// TIA Portal V16 export
// export: Created 2021-11-12T13:33:14.2128185Z, ExportSetting WithDefaults, DisplayName Totally Integrated Automation Portal, DisplayVersion V16 Update 3, DisplayName TIA Portal Version Control Interface, DisplayVersion V16 Update 2, DisplayName TIA Portal Openness, DisplayVersion V16 Update 3, DisplayName SINAMICS Startdrive Advanced, DisplayVersion V16 Update 5, DisplayName SINAMICS Startdrive G130, G150, S120, S150, SINAMICS MV, S210, DisplayVersion V16 Update 5, DisplayName SINAMICS Startdrive G110M, G120, G120C, G120D, G120P, G115D, DisplayVersion V16 Update 5, DisplayName STEP 7 Professional, DisplayVersion V16 Update 3, DisplayName STEP 7 Safety, DisplayVersion V16, DisplayName WinCC UA Professional, DisplayVersion V16 Update 3
FUNCTION_BLOCK "IM_400+UH31-KF10"   // FB24, LAD
TITLE = Inputs reading
{ S7_Optimized_Access := 'TRUE' }
VERSION : 0.1
// MICE Wood interface block
// stored: AutoNumber true, IsIECCheckEnabled false, IsRetainMemResEnabled false, MemoryReserve 100, SetENOAutomatically false, UDAEnableTagReadback false
   VAR
      KF11_Ix0 { S7_SetPoint := 'True'} : "STD_CH_DI";
      KF11_Ix1 { S7_SetPoint := 'True'} : "STD_CH_DI";
      KF11_Ix2 { S7_SetPoint := 'True'} : "STD_CH_DI";
      KF11_Ix3 { S7_SetPoint := 'True'} : "STD_CH_DI";
      KF11_Ix4 { S7_SetPoint := 'True'} : "STD_CH_DI";
      KF11_Ix5 { S7_SetPoint := 'True'} : "STD_CH_DI";
      KF11_Ix6 { S7_SetPoint := 'True'} : "STD_CH_DI";
      KF11_Ix7 { S7_SetPoint := 'True'} : "STD_CH_DI";
      KF12_Ix0 { S7_SetPoint := 'True'} : "STD_CH_DI";
      KF12_Ix1 { S7_SetPoint := 'True'} : "STD_CH_DI";
      KF12_Ix2 { S7_SetPoint := 'True'} : "STD_CH_DI";
      KF12_Ix3 { S7_SetPoint := 'True'} : "STD_CH_DI";
      KF12_Ix4 { S7_SetPoint := 'True'} : "STD_CH_DI";
      KF12_Ix5 { S7_SetPoint := 'True'} : "STD_CH_DI";
      KF12_Ix6 { S7_SetPoint := 'True'} : "STD_CH_DI";
      KF12_Ix7 { S7_SetPoint := 'True'} : "STD_CH_DI";
      KF12_Ix8 { S7_SetPoint := 'True'} : "STD_CH_DI";
      KF12_Ix9 { S7_SetPoint := 'True'} : "STD_CH_DI";
      KF12_Ix10 { S7_SetPoint := 'True'} : "STD_CH_DI";
      KF12_Ix11 { S7_SetPoint := 'True'} : "STD_CH_DI";
      KF12_Ix12 { S7_SetPoint := 'True'} : "STD_CH_DI";
      KF12_Ix13 { S7_SetPoint := 'True'} : "STD_CH_DI";
      KF12_Ix14 { S7_SetPoint := 'True'} : "STD_CH_DI";
      KF12_Ix15 { S7_SetPoint := 'True'} : "STD_CH_DI";
      KF13_Ix0 { S7_SetPoint := 'True'} : "STD_CH_DI";
      KF13_Ix1 { S7_SetPoint := 'True'} : "STD_CH_DI";
      KF13_Ix2 { S7_SetPoint := 'True'} : "STD_CH_DI";
      KF13_Ix3 { S7_SetPoint := 'True'} : "STD_CH_DI";
      KF13_Ix4 { S7_SetPoint := 'True'} : "STD_CH_DI";
      KF13_Ix5 { S7_SetPoint := 'True'} : "STD_CH_DI";
      KF13_Ix6 { S7_SetPoint := 'True'} : "STD_CH_DI";
      KF13_Ix7 { S7_SetPoint := 'True'} : "STD_CH_DI";
      KF13_Ix8 { S7_SetPoint := 'True'} : "STD_CH_DI";
      KF13_Ix9 { S7_SetPoint := 'True'} : "STD_CH_DI";
      KF13_Ix10 { S7_SetPoint := 'True'} : "STD_CH_DI";
      KF13_Ix11 { S7_SetPoint := 'True'} : "STD_CH_DI";
      KF13_Ix12 { S7_SetPoint := 'True'} : "STD_CH_DI";
      KF13_Ix13 { S7_SetPoint := 'True'} : "STD_CH_DI";
      KF13_Ix14 { S7_SetPoint := 'True'} : "STD_CH_DI";
      KF13_Ix15 { S7_SetPoint := 'True'} : "STD_CH_DI";
      KF14_Ix0 { S7_SetPoint := 'True'} : "STD_CH_DI";
      KF14_Ix1 { S7_SetPoint := 'True'} : "STD_CH_DI";
      KF14_Ix2 { S7_SetPoint := 'True'} : "STD_CH_DI";
      KF14_Ix3 { S7_SetPoint := 'True'} : "STD_CH_DI";
      KF14_Ix4 { S7_SetPoint := 'True'} : "STD_CH_DI";
      KF14_Ix5 { S7_SetPoint := 'True'} : "STD_CH_DI";
      KF14_Ix6 { S7_SetPoint := 'True'} : "STD_CH_DI";
      KF14_Ix7 { S7_SetPoint := 'True'} : "STD_CH_DI";
      KF14_Ix8 { S7_SetPoint := 'True'} : "STD_CH_DI";
      KF14_Ix9 { S7_SetPoint := 'True'} : "STD_CH_DI";
      KF14_Ix10 { S7_SetPoint := 'True'} : "STD_CH_DI";
      KF14_Ix11 { S7_SetPoint := 'True'} : "STD_CH_DI";
      KF14_Ix12 { S7_SetPoint := 'True'} : "STD_CH_DI";
      KF14_Ix13 { S7_SetPoint := 'True'} : "STD_CH_DI";
      KF14_Ix14 { S7_SetPoint := 'True'} : "STD_CH_DI";
      KF14_Ix15 { S7_SetPoint := 'True'} : "STD_CH_DI";
      KF15_Ix0 { S7_SetPoint := 'True'} : "STD_CH_DI";
      KF15_Ix1 { S7_SetPoint := 'True'} : "STD_CH_DI";
      KF15_Ix2 { S7_SetPoint := 'True'} : "STD_CH_DI";
      KF15_Ix3 { S7_SetPoint := 'True'} : "STD_CH_DI";
      KF15_Ix4 { S7_SetPoint := 'True'} : "STD_CH_DI";
      KF15_Ix5 { S7_SetPoint := 'True'} : "STD_CH_DI";
      KF15_Ix6 { S7_SetPoint := 'True'} : "STD_CH_DI";
      KF15_Ix7 { S7_SetPoint := 'True'} : "STD_CH_DI";
      KF15_Ix8 { S7_SetPoint := 'True'} : "STD_CH_DI";
      KF15_Ix9 { S7_SetPoint := 'True'} : "STD_CH_DI";
      KF15_Ix10 { S7_SetPoint := 'True'} : "STD_CH_DI";
      KF15_Ix11 { S7_SetPoint := 'True'} : "STD_CH_DI";
      KF15_Ix12 { S7_SetPoint := 'True'} : "STD_CH_DI";
      KF15_Ix13 { S7_SetPoint := 'True'} : "STD_CH_DI";
      KF15_Ix14 { S7_SetPoint := 'True'} : "STD_CH_DI";
      KF15_Ix15 { S7_SetPoint := 'True'} : "STD_CH_DI";
      KF61_AI0 { S7_SetPoint := 'True'} : "STD_CH_AI";
      KF61_AI1 { S7_SetPoint := 'True'} : "STD_CH_AI";
      KF61_AI2 { S7_SetPoint := 'True'} : "STD_CH_AI";
      KF61_AI3 { S7_SetPoint := 'True'} : "STD_CH_AI";
   END_VAR
   VAR_TEMP   // added for the SCL form of the ladder/FBD networks
      _w1 : Bool;
      _w2 : Bool;
      _w3 : Bool;
      _w4 : Bool;
      _w5 : Bool;
      _w6 : Bool;
      _w7 : Bool;
      _w8 : Bool;
   END_VAR
BEGIN

REGION Network 1: Module position -KF11
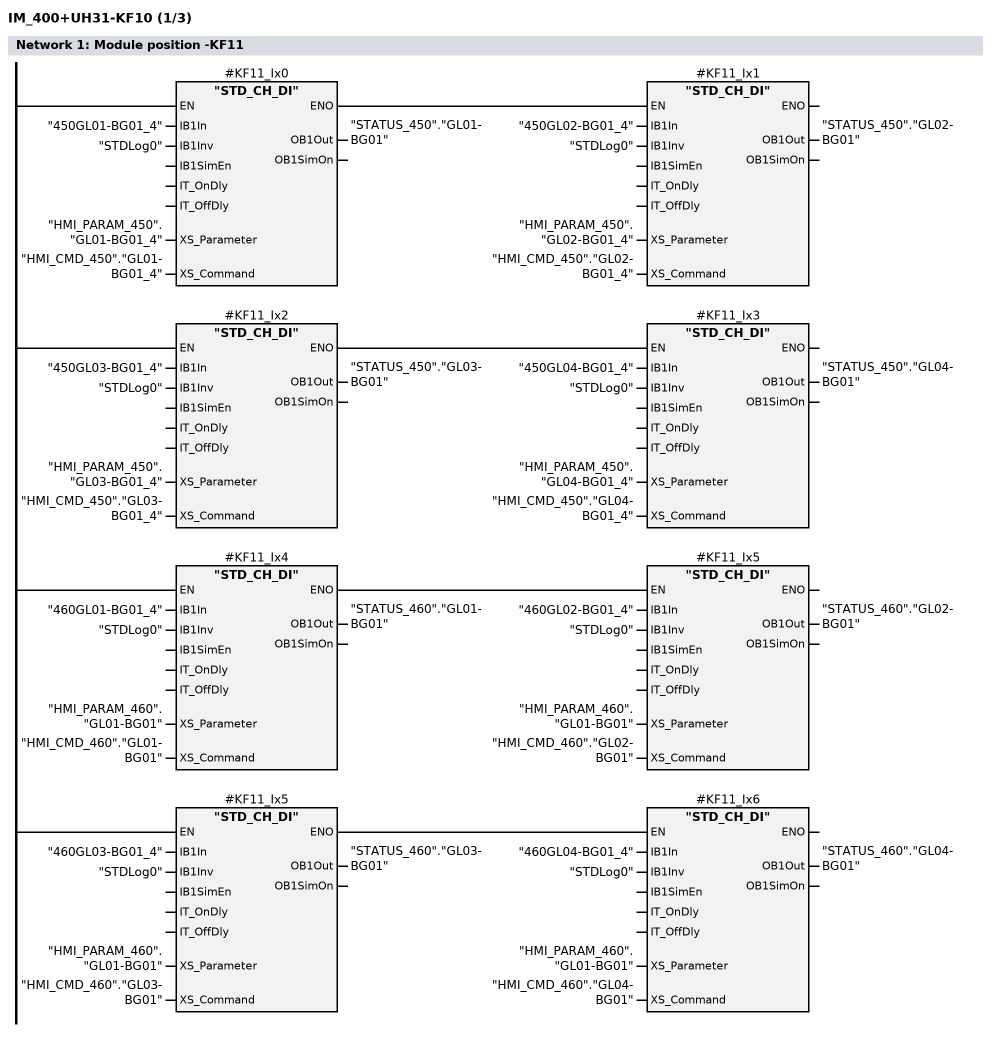
   RUNG wire#powerrail
      #KF11_Ix0(IB1In := "450GL01-BG01_4", IB1Inv := "STDLog0", IB1SimEn :=, IT_OnDly :=, IT_OffDly :=, XS_Parameter := "HMI_PARAM_450"."GL01-BG01_4", XS_Command := "HMI_CMD_450"."GL01-BG01_4", OB1Out => "STATUS_450"."GL01-BG01", OB1SimOn =>)
      #KF11_Ix1(IB1In := "450GL02-BG01_4", IB1Inv := "STDLog0", IB1SimEn :=, IT_OnDly :=, IT_OffDly :=, XS_Parameter := "HMI_PARAM_450"."GL02-BG01_4", XS_Command := "HMI_CMD_450"."GL02-BG01_4", OB1Out => "STATUS_450"."GL02-BG01", OB1SimOn =>)
   END_RUNG
   RUNG wire#powerrail
      #KF11_Ix2(IB1In := "450GL03-BG01_4", IB1Inv := "STDLog0", IB1SimEn :=, IT_OnDly :=, IT_OffDly :=, XS_Parameter := "HMI_PARAM_450"."GL03-BG01_4", XS_Command := "HMI_CMD_450"."GL03-BG01_4", OB1Out => "STATUS_450"."GL03-BG01", OB1SimOn =>)
      #KF11_Ix3(IB1In := "450GL04-BG01_4", IB1Inv := "STDLog0", IB1SimEn :=, IT_OnDly :=, IT_OffDly :=, XS_Parameter := "HMI_PARAM_450"."GL04-BG01_4", XS_Command := "HMI_CMD_450"."GL04-BG01_4", OB1Out => "STATUS_450"."GL04-BG01", OB1SimOn =>)
   END_RUNG
   RUNG wire#powerrail
      #KF11_Ix4(IB1In := "460GL01-BG01_4", IB1Inv := "STDLog0", IB1SimEn :=, IT_OnDly :=, IT_OffDly :=, XS_Parameter := "HMI_PARAM_460"."GL01-BG01", XS_Command := "HMI_CMD_460"."GL01-BG01", OB1Out => "STATUS_460"."GL01-BG01", OB1SimOn =>)
      #KF11_Ix5(IB1In := "460GL02-BG01_4", IB1Inv := "STDLog0", IB1SimEn :=, IT_OnDly :=, IT_OffDly :=, XS_Parameter := "HMI_PARAM_460"."GL01-BG01", XS_Command := "HMI_CMD_460"."GL02-BG01", OB1Out => "STATUS_460"."GL02-BG01", OB1SimOn =>)
   END_RUNG
   RUNG wire#powerrail
      #KF11_Ix5(IB1In := "460GL03-BG01_4", IB1Inv := "STDLog0", IB1SimEn :=, IT_OnDly :=, IT_OffDly :=, XS_Parameter := "HMI_PARAM_460"."GL01-BG01", XS_Command := "HMI_CMD_460"."GL03-BG01", OB1Out => "STATUS_460"."GL03-BG01", OB1SimOn =>)
      #KF11_Ix6(IB1In := "460GL04-BG01_4", IB1Inv := "STDLog0", IB1SimEn :=, IT_OnDly :=, IT_OffDly :=, XS_Parameter := "HMI_PARAM_460"."GL01-BG01", XS_Command := "HMI_CMD_460"."GL04-BG01", OB1Out => "STATUS_460"."GL04-BG01", OB1SimOn =>)
   END_RUNG
   // the same network as SCL:
   #KF11_Ix0(IB1In := "450GL01-BG01_4",   // "STD_CH_DI"
             IB1Inv := "STDLog0",
             XS_Parameter := "HMI_PARAM_450"."GL01-BG01_4",
             XS_Command := "HMI_CMD_450"."GL01-BG01_4",
             OB1Out => "STATUS_450"."GL01-BG01",
             ENO => #_w1);
   IF #_w1 THEN
       #KF11_Ix1(IB1In := "450GL02-BG01_4",   // "STD_CH_DI"
                 IB1Inv := "STDLog0",
                 XS_Parameter := "HMI_PARAM_450"."GL02-BG01_4",
                 XS_Command := "HMI_CMD_450"."GL02-BG01_4",
                 OB1Out => "STATUS_450"."GL02-BG01");
   END_IF;
   #KF11_Ix2(IB1In := "450GL03-BG01_4",   // "STD_CH_DI"
             IB1Inv := "STDLog0",
             XS_Parameter := "HMI_PARAM_450"."GL03-BG01_4",
             XS_Command := "HMI_CMD_450"."GL03-BG01_4",
             OB1Out => "STATUS_450"."GL03-BG01",
             ENO => #_w2);
   IF #_w2 THEN
       #KF11_Ix3(IB1In := "450GL04-BG01_4",   // "STD_CH_DI"
                 IB1Inv := "STDLog0",
                 XS_Parameter := "HMI_PARAM_450"."GL04-BG01_4",
                 XS_Command := "HMI_CMD_450"."GL04-BG01_4",
                 OB1Out => "STATUS_450"."GL04-BG01");
   END_IF;
   #KF11_Ix4(IB1In := "460GL01-BG01_4",   // "STD_CH_DI"
             IB1Inv := "STDLog0",
             XS_Parameter := "HMI_PARAM_460"."GL01-BG01",
             XS_Command := "HMI_CMD_460"."GL01-BG01",
             OB1Out => "STATUS_460"."GL01-BG01",
             ENO => #_w3);
   IF #_w3 THEN
       #KF11_Ix5(IB1In := "460GL02-BG01_4",   // "STD_CH_DI"
                 IB1Inv := "STDLog0",
                 XS_Parameter := "HMI_PARAM_460"."GL01-BG01",
                 XS_Command := "HMI_CMD_460"."GL02-BG01",
                 OB1Out => "STATUS_460"."GL02-BG01");
   END_IF;
   #KF11_Ix5(IB1In := "460GL03-BG01_4",   // "STD_CH_DI"
             IB1Inv := "STDLog0",
             XS_Parameter := "HMI_PARAM_460"."GL01-BG01",
             XS_Command := "HMI_CMD_460"."GL03-BG01",
             OB1Out => "STATUS_460"."GL03-BG01",
             ENO => #_w4);
   IF #_w4 THEN
       #KF11_Ix6(IB1In := "460GL04-BG01_4",   // "STD_CH_DI"
                 IB1Inv := "STDLog0",
                 XS_Parameter := "HMI_PARAM_460"."GL01-BG01",
                 XS_Command := "HMI_CMD_460"."GL04-BG01",
                 OB1Out => "STATUS_460"."GL04-BG01");
   END_IF;
END_REGION

REGION Network 2: Module position -kf12
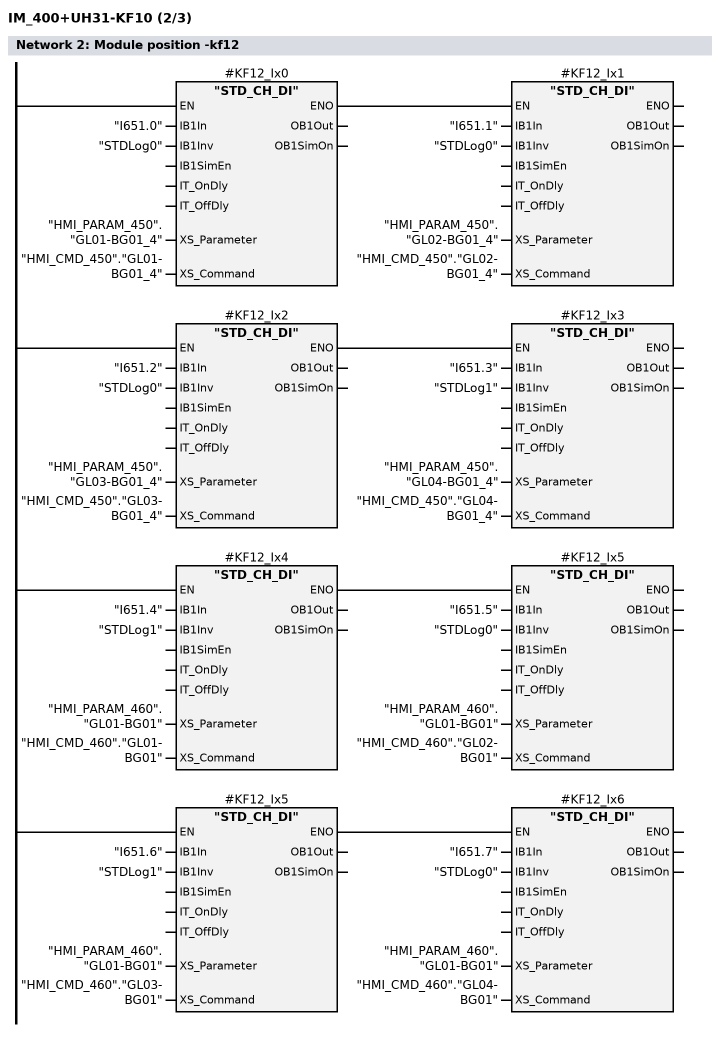
   RUNG wire#powerrail
      #KF12_Ix0(IB1In := "I651.0", IB1Inv := "STDLog0", IB1SimEn :=, IT_OnDly :=, IT_OffDly :=, XS_Parameter := "HMI_PARAM_450"."GL01-BG01_4", XS_Command := "HMI_CMD_450"."GL01-BG01_4", OB1Out =>, OB1SimOn =>)
      #KF12_Ix1(IB1In := "I651.1", IB1Inv := "STDLog0", IB1SimEn :=, IT_OnDly :=, IT_OffDly :=, XS_Parameter := "HMI_PARAM_450"."GL02-BG01_4", XS_Command := "HMI_CMD_450"."GL02-BG01_4", OB1Out =>, OB1SimOn =>)
   END_RUNG
   RUNG wire#powerrail
      #KF12_Ix2(IB1In := "I651.2", IB1Inv := "STDLog0", IB1SimEn :=, IT_OnDly :=, IT_OffDly :=, XS_Parameter := "HMI_PARAM_450"."GL03-BG01_4", XS_Command := "HMI_CMD_450"."GL03-BG01_4", OB1Out =>, OB1SimOn =>)
      #KF12_Ix3(IB1In := "I651.3", IB1Inv := "STDLog1", IB1SimEn :=, IT_OnDly :=, IT_OffDly :=, XS_Parameter := "HMI_PARAM_450"."GL04-BG01_4", XS_Command := "HMI_CMD_450"."GL04-BG01_4", OB1Out =>, OB1SimOn =>)
   END_RUNG
   RUNG wire#powerrail
      #KF12_Ix4(IB1In := "I651.4", IB1Inv := "STDLog1", IB1SimEn :=, IT_OnDly :=, IT_OffDly :=, XS_Parameter := "HMI_PARAM_460"."GL01-BG01", XS_Command := "HMI_CMD_460"."GL01-BG01", OB1Out =>, OB1SimOn =>)
      #KF12_Ix5(IB1In := "I651.5", IB1Inv := "STDLog0", IB1SimEn :=, IT_OnDly :=, IT_OffDly :=, XS_Parameter := "HMI_PARAM_460"."GL01-BG01", XS_Command := "HMI_CMD_460"."GL02-BG01", OB1Out =>, OB1SimOn =>)
   END_RUNG
   RUNG wire#powerrail
      #KF12_Ix5(IB1In := "I651.6", IB1Inv := "STDLog1", IB1SimEn :=, IT_OnDly :=, IT_OffDly :=, XS_Parameter := "HMI_PARAM_460"."GL01-BG01", XS_Command := "HMI_CMD_460"."GL03-BG01", OB1Out =>, OB1SimOn =>)
      #KF12_Ix6(IB1In := "I651.7", IB1Inv := "STDLog0", IB1SimEn :=, IT_OnDly :=, IT_OffDly :=, XS_Parameter := "HMI_PARAM_460"."GL01-BG01", XS_Command := "HMI_CMD_460"."GL04-BG01", OB1Out =>, OB1SimOn =>)
   END_RUNG
   // the same network as SCL:
   #KF12_Ix0(IB1In := "I651.0",   // "STD_CH_DI"
             IB1Inv := "STDLog0",
             XS_Parameter := "HMI_PARAM_450"."GL01-BG01_4",
             XS_Command := "HMI_CMD_450"."GL01-BG01_4",
             ENO => #_w1);
   IF #_w1 THEN
       #KF12_Ix1(IB1In := "I651.1",   // "STD_CH_DI"
                 IB1Inv := "STDLog0",
                 XS_Parameter := "HMI_PARAM_450"."GL02-BG01_4",
                 XS_Command := "HMI_CMD_450"."GL02-BG01_4");
   END_IF;
   #KF12_Ix2(IB1In := "I651.2",   // "STD_CH_DI"
             IB1Inv := "STDLog0",
             XS_Parameter := "HMI_PARAM_450"."GL03-BG01_4",
             XS_Command := "HMI_CMD_450"."GL03-BG01_4",
             ENO => #_w2);
   IF #_w2 THEN
       #KF12_Ix3(IB1In := "I651.3",   // "STD_CH_DI"
                 IB1Inv := "STDLog1",
                 XS_Parameter := "HMI_PARAM_450"."GL04-BG01_4",
                 XS_Command := "HMI_CMD_450"."GL04-BG01_4");
   END_IF;
   #KF12_Ix4(IB1In := "I651.4",   // "STD_CH_DI"
             IB1Inv := "STDLog1",
             XS_Parameter := "HMI_PARAM_460"."GL01-BG01",
             XS_Command := "HMI_CMD_460"."GL01-BG01",
             ENO => #_w3);
   IF #_w3 THEN
       #KF12_Ix5(IB1In := "I651.5",   // "STD_CH_DI"
                 IB1Inv := "STDLog0",
                 XS_Parameter := "HMI_PARAM_460"."GL01-BG01",
                 XS_Command := "HMI_CMD_460"."GL02-BG01");
   END_IF;
   #KF12_Ix5(IB1In := "I651.6",   // "STD_CH_DI"
             IB1Inv := "STDLog1",
             XS_Parameter := "HMI_PARAM_460"."GL01-BG01",
             XS_Command := "HMI_CMD_460"."GL03-BG01",
             ENO => #_w4);
   IF #_w4 THEN
       #KF12_Ix6(IB1In := "I651.7",   // "STD_CH_DI"
                 IB1Inv := "STDLog0",
                 XS_Parameter := "HMI_PARAM_460"."GL01-BG01",
                 XS_Command := "HMI_CMD_460"."GL04-BG01");
   END_IF;
END_REGION

REGION Network 3: Module position -KF13
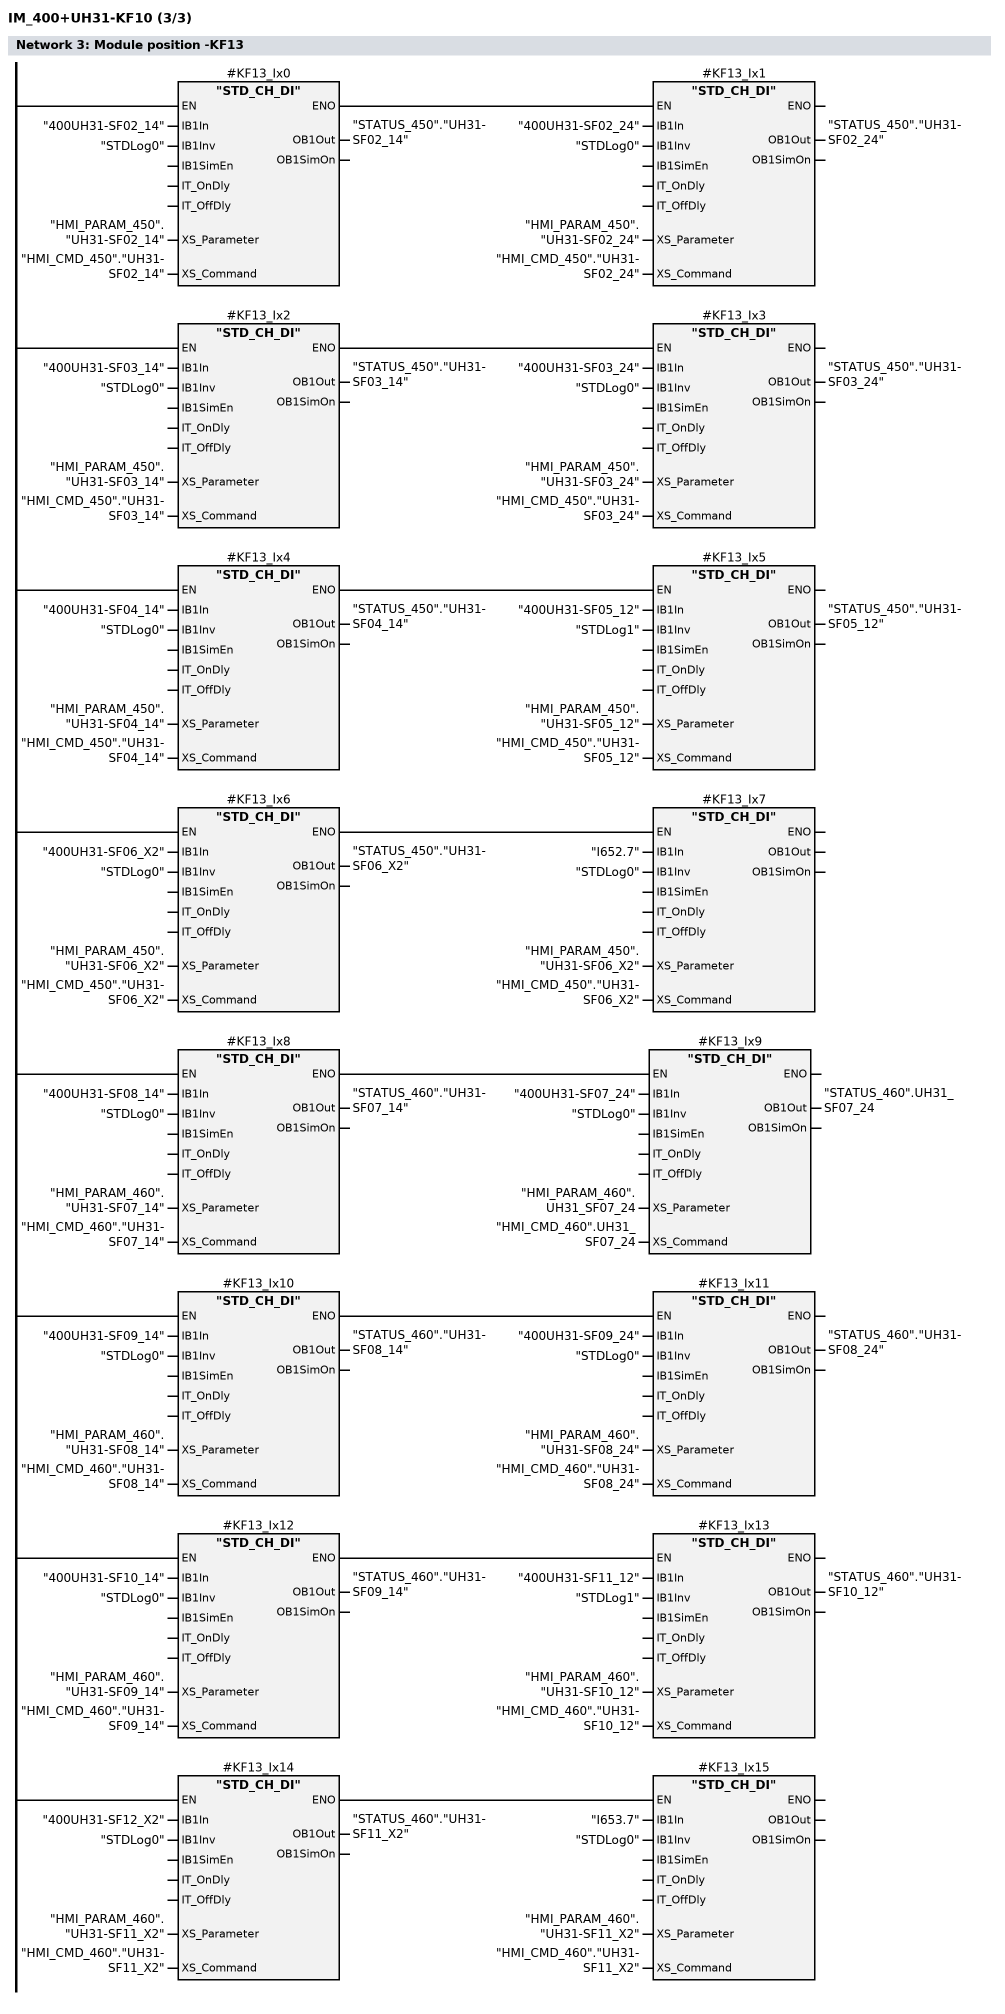
   RUNG wire#powerrail
      #KF13_Ix0(IB1In := "400UH31-SF02_14", IB1Inv := "STDLog0", IB1SimEn :=, IT_OnDly :=, IT_OffDly :=, XS_Parameter := "HMI_PARAM_450"."UH31-SF02_14", XS_Command := "HMI_CMD_450"."UH31-SF02_14", OB1Out => "STATUS_450"."UH31-SF02_14", OB1SimOn =>)
      #KF13_Ix1(IB1In := "400UH31-SF02_24", IB1Inv := "STDLog0", IB1SimEn :=, IT_OnDly :=, IT_OffDly :=, XS_Parameter := "HMI_PARAM_450"."UH31-SF02_24", XS_Command := "HMI_CMD_450"."UH31-SF02_24", OB1Out => "STATUS_450"."UH31-SF02_24", OB1SimOn =>)
   END_RUNG
   RUNG wire#powerrail
      #KF13_Ix2(IB1In := "400UH31-SF03_14", IB1Inv := "STDLog0", IB1SimEn :=, IT_OnDly :=, IT_OffDly :=, XS_Parameter := "HMI_PARAM_450"."UH31-SF03_14", XS_Command := "HMI_CMD_450"."UH31-SF03_14", OB1Out => "STATUS_450"."UH31-SF03_14", OB1SimOn =>)
      #KF13_Ix3(IB1In := "400UH31-SF03_24", IB1Inv := "STDLog0", IB1SimEn :=, IT_OnDly :=, IT_OffDly :=, XS_Parameter := "HMI_PARAM_450"."UH31-SF03_24", XS_Command := "HMI_CMD_450"."UH31-SF03_24", OB1Out => "STATUS_450"."UH31-SF03_24", OB1SimOn =>)
   END_RUNG
   RUNG wire#powerrail
      #KF13_Ix4(IB1In := "400UH31-SF04_14", IB1Inv := "STDLog0", IB1SimEn :=, IT_OnDly :=, IT_OffDly :=, XS_Parameter := "HMI_PARAM_450"."UH31-SF04_14", XS_Command := "HMI_CMD_450"."UH31-SF04_14", OB1Out => "STATUS_450"."UH31-SF04_14", OB1SimOn =>)
      #KF13_Ix5(IB1In := "400UH31-SF05_12", IB1Inv := "STDLog1", IB1SimEn :=, IT_OnDly :=, IT_OffDly :=, XS_Parameter := "HMI_PARAM_450"."UH31-SF05_12", XS_Command := "HMI_CMD_450"."UH31-SF05_12", OB1Out => "STATUS_450"."UH31-SF05_12", OB1SimOn =>)
   END_RUNG
   RUNG wire#powerrail
      #KF13_Ix6(IB1In := "400UH31-SF06_X2", IB1Inv := "STDLog0", IB1SimEn :=, IT_OnDly :=, IT_OffDly :=, XS_Parameter := "HMI_PARAM_450"."UH31-SF06_X2", XS_Command := "HMI_CMD_450"."UH31-SF06_X2", OB1Out => "STATUS_450"."UH31-SF06_X2", OB1SimOn =>)
      #KF13_Ix7(IB1In := "I652.7", IB1Inv := "STDLog0", IB1SimEn :=, IT_OnDly :=, IT_OffDly :=, XS_Parameter := "HMI_PARAM_450"."UH31-SF06_X2", XS_Command := "HMI_CMD_450"."UH31-SF06_X2", OB1Out =>, OB1SimOn =>)
   END_RUNG
   RUNG wire#powerrail
      #KF13_Ix8(IB1In := "400UH31-SF08_14", IB1Inv := "STDLog0", IB1SimEn :=, IT_OnDly :=, IT_OffDly :=, XS_Parameter := "HMI_PARAM_460"."UH31-SF07_14", XS_Command := "HMI_CMD_460"."UH31-SF07_14", OB1Out => "STATUS_460"."UH31-SF07_14", OB1SimOn =>)
      #KF13_Ix9(IB1In := "400UH31-SF07_24", IB1Inv := "STDLog0", IB1SimEn :=, IT_OnDly :=, IT_OffDly :=, XS_Parameter := "HMI_PARAM_460".UH31_SF07_24, XS_Command := "HMI_CMD_460".UH31_SF07_24, OB1Out => "STATUS_460".UH31_SF07_24, OB1SimOn =>)
   END_RUNG
   RUNG wire#powerrail
      #KF13_Ix10(IB1In := "400UH31-SF09_14", IB1Inv := "STDLog0", IB1SimEn :=, IT_OnDly :=, IT_OffDly :=, XS_Parameter := "HMI_PARAM_460"."UH31-SF08_14", XS_Command := "HMI_CMD_460"."UH31-SF08_14", OB1Out => "STATUS_460"."UH31-SF08_14", OB1SimOn =>)
      #KF13_Ix11(IB1In := "400UH31-SF09_24", IB1Inv := "STDLog0", IB1SimEn :=, IT_OnDly :=, IT_OffDly :=, XS_Parameter := "HMI_PARAM_460"."UH31-SF08_24", XS_Command := "HMI_CMD_460"."UH31-SF08_24", OB1Out => "STATUS_460"."UH31-SF08_24", OB1SimOn =>)
   END_RUNG
   RUNG wire#powerrail
      #KF13_Ix12(IB1In := "400UH31-SF10_14", IB1Inv := "STDLog0", IB1SimEn :=, IT_OnDly :=, IT_OffDly :=, XS_Parameter := "HMI_PARAM_460"."UH31-SF09_14", XS_Command := "HMI_CMD_460"."UH31-SF09_14", OB1Out => "STATUS_460"."UH31-SF09_14", OB1SimOn =>)
      #KF13_Ix13(IB1In := "400UH31-SF11_12", IB1Inv := "STDLog1", IB1SimEn :=, IT_OnDly :=, IT_OffDly :=, XS_Parameter := "HMI_PARAM_460"."UH31-SF10_12", XS_Command := "HMI_CMD_460"."UH31-SF10_12", OB1Out => "STATUS_460"."UH31-SF10_12", OB1SimOn =>)
   END_RUNG
   RUNG wire#powerrail
      #KF13_Ix14(IB1In := "400UH31-SF12_X2", IB1Inv := "STDLog0", IB1SimEn :=, IT_OnDly :=, IT_OffDly :=, XS_Parameter := "HMI_PARAM_460"."UH31-SF11_X2", XS_Command := "HMI_CMD_460"."UH31-SF11_X2", OB1Out => "STATUS_460"."UH31-SF11_X2", OB1SimOn =>)
      #KF13_Ix15(IB1In := "I653.7", IB1Inv := "STDLog0", IB1SimEn :=, IT_OnDly :=, IT_OffDly :=, XS_Parameter := "HMI_PARAM_460"."UH31-SF11_X2", XS_Command := "HMI_CMD_460"."UH31-SF11_X2", OB1Out =>, OB1SimOn =>)
   END_RUNG
   // the same network as SCL:
   #KF13_Ix0(IB1In := "400UH31-SF02_14",   // "STD_CH_DI"
             IB1Inv := "STDLog0",
             XS_Parameter := "HMI_PARAM_450"."UH31-SF02_14",
             XS_Command := "HMI_CMD_450"."UH31-SF02_14",
             OB1Out => "STATUS_450"."UH31-SF02_14",
             ENO => #_w1);
   IF #_w1 THEN
       #KF13_Ix1(IB1In := "400UH31-SF02_24",   // "STD_CH_DI"
                 IB1Inv := "STDLog0",
                 XS_Parameter := "HMI_PARAM_450"."UH31-SF02_24",
                 XS_Command := "HMI_CMD_450"."UH31-SF02_24",
                 OB1Out => "STATUS_450"."UH31-SF02_24");
   END_IF;
   #KF13_Ix2(IB1In := "400UH31-SF03_14",   // "STD_CH_DI"
             IB1Inv := "STDLog0",
             XS_Parameter := "HMI_PARAM_450"."UH31-SF03_14",
             XS_Command := "HMI_CMD_450"."UH31-SF03_14",
             OB1Out => "STATUS_450"."UH31-SF03_14",
             ENO => #_w2);
   IF #_w2 THEN
       #KF13_Ix3(IB1In := "400UH31-SF03_24",   // "STD_CH_DI"
                 IB1Inv := "STDLog0",
                 XS_Parameter := "HMI_PARAM_450"."UH31-SF03_24",
                 XS_Command := "HMI_CMD_450"."UH31-SF03_24",
                 OB1Out => "STATUS_450"."UH31-SF03_24");
   END_IF;
   #KF13_Ix4(IB1In := "400UH31-SF04_14",   // "STD_CH_DI"
             IB1Inv := "STDLog0",
             XS_Parameter := "HMI_PARAM_450"."UH31-SF04_14",
             XS_Command := "HMI_CMD_450"."UH31-SF04_14",
             OB1Out => "STATUS_450"."UH31-SF04_14",
             ENO => #_w3);
   IF #_w3 THEN
       #KF13_Ix5(IB1In := "400UH31-SF05_12",   // "STD_CH_DI"
                 IB1Inv := "STDLog1",
                 XS_Parameter := "HMI_PARAM_450"."UH31-SF05_12",
                 XS_Command := "HMI_CMD_450"."UH31-SF05_12",
                 OB1Out => "STATUS_450"."UH31-SF05_12");
   END_IF;
   #KF13_Ix6(IB1In := "400UH31-SF06_X2",   // "STD_CH_DI"
             IB1Inv := "STDLog0",
             XS_Parameter := "HMI_PARAM_450"."UH31-SF06_X2",
             XS_Command := "HMI_CMD_450"."UH31-SF06_X2",
             OB1Out => "STATUS_450"."UH31-SF06_X2",
             ENO => #_w4);
   IF #_w4 THEN
       #KF13_Ix7(IB1In := "I652.7",   // "STD_CH_DI"
                 IB1Inv := "STDLog0",
                 XS_Parameter := "HMI_PARAM_450"."UH31-SF06_X2",
                 XS_Command := "HMI_CMD_450"."UH31-SF06_X2");
   END_IF;
   #KF13_Ix8(IB1In := "400UH31-SF08_14",   // "STD_CH_DI"
             IB1Inv := "STDLog0",
             XS_Parameter := "HMI_PARAM_460"."UH31-SF07_14",
             XS_Command := "HMI_CMD_460"."UH31-SF07_14",
             OB1Out => "STATUS_460"."UH31-SF07_14",
             ENO => #_w5);
   IF #_w5 THEN
       #KF13_Ix9(IB1In := "400UH31-SF07_24",   // "STD_CH_DI"
                 IB1Inv := "STDLog0",
                 XS_Parameter := "HMI_PARAM_460".UH31_SF07_24,
                 XS_Command := "HMI_CMD_460".UH31_SF07_24,
                 OB1Out => "STATUS_460".UH31_SF07_24);
   END_IF;
   #KF13_Ix10(IB1In := "400UH31-SF09_14",   // "STD_CH_DI"
              IB1Inv := "STDLog0",
              XS_Parameter := "HMI_PARAM_460"."UH31-SF08_14",
              XS_Command := "HMI_CMD_460"."UH31-SF08_14",
              OB1Out => "STATUS_460"."UH31-SF08_14",
              ENO => #_w6);
   IF #_w6 THEN
       #KF13_Ix11(IB1In := "400UH31-SF09_24",   // "STD_CH_DI"
                  IB1Inv := "STDLog0",
                  XS_Parameter := "HMI_PARAM_460"."UH31-SF08_24",
                  XS_Command := "HMI_CMD_460"."UH31-SF08_24",
                  OB1Out => "STATUS_460"."UH31-SF08_24");
   END_IF;
   #KF13_Ix12(IB1In := "400UH31-SF10_14",   // "STD_CH_DI"
              IB1Inv := "STDLog0",
              XS_Parameter := "HMI_PARAM_460"."UH31-SF09_14",
              XS_Command := "HMI_CMD_460"."UH31-SF09_14",
              OB1Out => "STATUS_460"."UH31-SF09_14",
              ENO => #_w7);
   IF #_w7 THEN
       #KF13_Ix13(IB1In := "400UH31-SF11_12",   // "STD_CH_DI"
                  IB1Inv := "STDLog1",
                  XS_Parameter := "HMI_PARAM_460"."UH31-SF10_12",
                  XS_Command := "HMI_CMD_460"."UH31-SF10_12",
                  OB1Out => "STATUS_460"."UH31-SF10_12");
   END_IF;
   #KF13_Ix14(IB1In := "400UH31-SF12_X2",   // "STD_CH_DI"
              IB1Inv := "STDLog0",
              XS_Parameter := "HMI_PARAM_460"."UH31-SF11_X2",
              XS_Command := "HMI_CMD_460"."UH31-SF11_X2",
              OB1Out => "STATUS_460"."UH31-SF11_X2",
              ENO => #_w8);
   IF #_w8 THEN
       #KF13_Ix15(IB1In := "I653.7",   // "STD_CH_DI"
                  IB1Inv := "STDLog0",
                  XS_Parameter := "HMI_PARAM_460"."UH31-SF11_X2",
                  XS_Command := "HMI_CMD_460"."UH31-SF11_X2");
   END_IF;
END_REGION
END_FUNCTION_BLOCK
